FUNCTION calculateTargetTemperatureOff : REAL
VAR_INPUT
	photovoltaicSurplus			: BOOL;
END_VAR

IF (photovoltaicSurplus) THEN
    calculateTargetTemperatureOff := GVL.configValues.targetTemperatureOffPV;
ELSE
    calculateTargetTemperatureOff := GVL.configValues.targetTemperatureOff;
END_IF;

END_FUNCTION

(* stored: Version 1.1.0.1
   POU calculateTargetTemperatureOff: Id {7db5afe6-c836-4eb4-8762-fc21a3ee7caa}, SpecialFunc None *)
